FUNCTION_BLOCK FB_Conveyor
VAR_INPUT
	sName					:STRING;
	bEn						:BOOL;				(*Enable - Engedély jel*)
	bEHA					:BOOL; 				(*Error-handling active - Hibafigyelés aktív*)
	bDisableManualCmd		:BOOL;				(*Manual control disable*)
	bConveyorOnL			:BOOL;				(*Control to Motor on - vezérlés parancs motor indításhoz*)
	bConveyorOnR			:BOOL;				(*Control to Motor on - vezérlés parancs motor indításhoz*)
	timReset				:TIME := T#2S;		(*Resettime - Hibatörlési idő*)
	bAck					:BOOL; 				(*Acknowledge - Hibanyugta*)
	i_bConveyorOK	AT %I*	:BOOL;				(*Conveyor drive OK - motorindító üzemkész*)
	stStartEvent			:TcEventEntry;		(*Event definition*)
	stRunEvent				:TcEventEntry;		(*Event definition*)
END_VAR
VAR_OUTPUT
	bMotorOn				:BOOL;				(* Motor on - Motor bekapcsolva *)
	bError					:BOOL;				(* Error bit - Hiba van *)
	sError					:STRING(255);		(* Error string - Hiba string *)
	q_bConveyorOnL	AT %Q*	:BOOL;				(* Motor on signal - Motor vezérlés bekapcsolása*)
	q_bConveyorOnR	AT %Q*	:BOOL;				(* Motor on signal - Motor vezérlés bekapcsolása*)
	q_bConveyorRst	AT %Q*	:BOOL;				(* Motor reset signal - Motor hibatörlés*)
END_VAR
VAR
	tMotorOn			:TON;
	tError,tFault		:TON;
	tReset				:TON;
	bErrOn,bErrRun		:BOOL;
	aErrorDesc			:ARRAY [0..1] OF STRING := [
	' motor hiba : a motorvezérlő nem indítható ', 
	' motor hiba : a motorvezérlő hibába van '];
	sEmpty				:STRING:='';
	bIsInitalized		:BOOL;
	fbStartAlarm		:FB_TcAlarm;
	fbRunAlarm			:FB_TcAlarm;
END_VAR

(*Hibanyugta*)
IF bAck OR NOT(bEHA) THEN
	bErrOn:=FALSE;
	bErrRun:=FALSE;
END_IF;

(* Motor bekapcsolási hiba *)
IF bEn AND bEHA AND (q_bConveyorOnL OR q_bConveyorOnR) AND NOT i_bConveyorOK THEN
	bErrOn:=TRUE;
	IF (fbStartAlarm.eConfirmationState <> 2 AND fbStartAlarm.nTimeCleared <> 0 AND fbStartAlarm.nTimeConfirmed <> 0) OR //Ha már volt alarm, akkor van bennük érték
		(fbStartAlarm.eConfirmationState = 1 AND fbStartAlarm.nTimeCleared = 0 AND fbStartAlarm.nTimeConfirmed = 0)	//Első futás esetén
	THEN
		fbStartAlarm.Raise(0);
	END_IF
END_IF;

(* Motor üzemzavar *)
tFault(IN:= bEn AND bEHA AND NOT i_bConveyorOK AND NOT bErrRun, PT:= T#5S);
IF tFault.Q THEN
	bErrRun:=TRUE;
	IF (fbRunAlarm.eConfirmationState <> 2 AND fbRunAlarm.nTimeCleared <> 0 AND fbRunAlarm.nTimeConfirmed <> 0) OR //Ha már volt alarm, akkor van bennük érték
		(fbRunAlarm.eConfirmationState = 1 AND fbRunAlarm.nTimeCleared = 0 AND fbRunAlarm.nTimeConfirmed = 0)	//Első futás esetén
	THEN
		fbRunAlarm.Raise(0);
	END_IF
END_IF;

(* Hibagyűjtő *)
bError := bErrOn OR bErrRun;

(*Vezérlés*)
IF 		bEn AND bConveyorOnL AND NOT bConveyorOnR AND i_bConveyorOK AND (NOT(bEHA) OR NOT(bError)) THEN
			q_bConveyorOnL := TRUE;
			q_bConveyorOnR := FALSE;
ELSIF	bEn AND NOT bConveyorOnL AND bConveyorOnR AND i_bConveyorOK AND (NOT(bEHA) OR NOT(bError)) THEN
			q_bConveyorOnL := FALSE;
			q_bConveyorOnR := TRUE;
ELSE
	q_bConveyorOnL := FALSE;
	q_bConveyorOnR := FALSE;
END_IF

(* Motor bekapcsolva *)
tMotorOn(IN:= (q_bConveyorOnL OR q_bConveyorOnR) AND NOT bError, 
	PT:= T#1S,
	Q=>  bMotorOn);

(* Manual reset *)
IF bError AND bAck AND NOT q_bConveyorRst THEN
	q_bConveyorRst := TRUE;
END_IF

tReset(IN:= q_bConveyorRst, PT:= timReset, Q=> , ET=> );
IF tReset.Q THEN
	q_bConveyorRst := FALSE;
END_IF

(*Hiba string*)
IF bErrOn OR bErrRun THEN
	sError := sName;
	IF bErrOn THEN
		sError :=  CONCAT(sError, aErrorDesc[0]);
	END_IF
	IF bErrRun THEN
		sError :=  CONCAT(sError, aErrorDesc[1]);
	END_IF
ELSE
	sError := sEmpty;
END_IF

(*Hiba kezelés Tc3_EventLogger*)
IF NOT bIsInitalized THEN
	bIsInitalized := TRUE;
	fbStartAlarm.CreateEx(stStartEvent, TRUE, 0);
	fbRunAlarm.CreateEx(stRunEvent, TRUE, 0);
END_IF

(*Hiba törlés (nyugtázott és megszűnt)*)
IF fbStartAlarm.eConfirmationState = 3 AND NOT bError THEN
	fbStartAlarm.Clear(0, FALSE);
END_IF	
IF fbRunAlarm.eConfirmationState = 3 AND NOT bError THEN
	fbRunAlarm.Clear(0, FALSE);
END_IF

END_FUNCTION_BLOCK

(* stored: Version 1.1.0.1, ProductVersion 3.1.4024.11
   POU FB_Conveyor: Id {68a09752-2bea-4d2f-a3eb-0138815d1853}, SpecialFunc None *)
